// TwinCAT 3 PLC project PLC1
// ProgramVersion: 3.1.4024.0
// libraries:
//   Tc2_ModbusRTU, * (Beckhoff Automation GmbH)
//   Tc2_Standard, * (Beckhoff Automation GmbH)
//   Tc2_System, * (Beckhoff Automation GmbH)
//   Tc3_Module, * (Beckhoff Automation GmbH)
// project tree:
//   / PlcTask.TcTTO
//   POUs/ MAIN.TcPOU
// real-time tasks:
//   TASK PlcTask: cycle T#10ms, priority 20, ADS port 350
// I/O:
//   DEVICE Device 1 (NOV-DP-RAM)
//   DEVICE Device 2 (CX7000), AmsNetId 5.132.90.65.3.1
//     Term 1 (CX7028) [CX7028-0000-0118]
//       modules: Module 1 (DIO_2x), Module 3 (DIO_2x), Module 5 (DI_2x), Module 7 (DI_2x)
//   DEVICE Device 3 (COM Port)
//   DEVICE Device 4 (COM Port)
// variable links:
//   PLC1/PLC1 Instance <-> Device 4 (COM Port)
//     PlcTask Inputs/MAIN.mbRTUMaster.InData/D <-> Inputs/Data1
//     PlcTask Inputs/MAIN.mbRTUMaster.InData/D @bit {8..504 step 8} <-> Inputs/Data{2..64}  (63 links)
//     PlcTask Inputs/MAIN.mbRTUMaster.InData/SerStatus <-> Inputs/Status
//     PlcTask Outputs/MAIN.mbRTUMaster.OutData/D <-> Outputs/Data1
//     PlcTask Outputs/MAIN.mbRTUMaster.OutData/D @bit {8..504 step 8} <-> Outputs/Data{2..64}  (63 links)
//     PlcTask Outputs/MAIN.mbRTUMaster.OutData/SerCtrl <-> Outputs/Ctrl

CONFIGURATION PLC1
    RESOURCE PLC ON TwinCAT3
        TASK PlcTask(INTERVAL := T#10ms, PRIORITY := 20);
        PROGRAM MAIN WITH PlcTask : MAIN;
    END_RESOURCE
END_CONFIGURATION

// ---- POUs/MAIN.TcPOU
PROGRAM MAIN
VAR
	mbRTUMaster			: ModbusRtuMaster_PcCOM;
	byMb_ID				: BYTE;
	wMb_ReadQtd			: WORD;
	wMb_ReadAddr		: WORD;
	arrData_Read		: ARRAY[1..10] OF INT;
	wData_Write			: WORD;
	bExecute			: BOOL;
	bExecute_Write		: BOOL;
END_VAR

mbRTUMaster.ReadRegs(
	UnitID:= byMb_ID, 
	Quantity:= wMb_ReadQtd, 
	MBAddr:= wMb_ReadAddr, 
	cbLength:= SIZEOF(arrData_Read), 
	pMemoryAddr:= ADR(arrData_Read), 
	Execute:= bExecute, 
	Timeout:= T#10S, 
	BUSY=> , 
	Error=> , 
	ErrorId=> , 
	cbRead=> );
	
	
mbRTUMaster.WriteRegs(
	UnitID:= byMb_ID, 
	Quantity:= 1,
	MBAddr:= wData_Write, 
	cbLength:= SIZEOF(wData_Write), 
	pMemoryAddr:= ADR(wData_Write), 
	Execute:= bExecute_Write, 
	Timeout:= T#10S, 
	BUSY=> , 
	Error=> , 
	ErrorId=> , 
	cbRead=> );

END_PROGRAM
